// TwinCAT 3 PLC project PLC1
// ProgramVersion: 3.1.4023.0
// libraries:
//   Tc2_Standard, * (Beckhoff Automation GmbH)
//   Tc2_System, * (Beckhoff Automation GmbH)
//   Tc3_Module, * (Beckhoff Automation GmbH)
// project tree:
//   / PlcTask.TcTTO
//   POUs/ MAIN.TcPOU

CONFIGURATION PLC1
    RESOURCE PLC ON TwinCAT3
        TASK PlcTask(INTERVAL := T#10ms, PRIORITY := 20);
        PROGRAM MAIN WITH PlcTask : MAIN;
    END_RESOURCE
END_CONFIGURATION

// ---- POUs/MAIN.TcPOU
PROGRAM MAIN
VAR
	Timer: ton;
	val: USINT := 0;
	nvar: usint := 0;
END_VAR

Timer(in:= NOT Timer.Q, pt:= T#0.5S);

IF (timer.Q) THEN
	val := val + 20;
	IF (val>100) THEN
		val := 0;
	END_IF
END_IF

nvar:=100-val;

END_PROGRAM
